Staubli VAL3: clkValve3.pgx

program clkValve3()
begin
  call toggleValve(3)
end
